// TIA Portal project "THAY PHUONG" (V17)

(* hardware
DEVICE "S7-1200 station_1"  S7-1200 Station
   slot 0: "Rack_0"  S7-1200 Rack  Rack  V1.0
   slot 1: "PLC_1"  CPU 1214C DC/DC/DC  6ES7 214-1AG40-0XB0  V4.0
*)

// ===== PLC "PLC_1"  CPU 1214C DC/DC/DC =====

VAR_GLOBAL   // PLC tag table "Default tag table"
   "System_Byte" AT %MB100 : Byte;
   "FirstScan" AT %M100.0 : Bool;
   "DiagStatusUpdate" AT %M100.1 : Bool;
   "AlwaysTRUE" AT %M100.2 : Bool;
   "AlwaysFALSE" AT %M100.3 : Bool;
   "Clock_Byte" AT %MB200 : Byte;
   "Clock_10Hz" AT %M200.0 : Bool;
   "Clock_5Hz" AT %M200.1 : Bool;
   "Clock_2.5Hz" AT %M200.2 : Bool;
   "Clock_2Hz" AT %M200.3 : Bool;
   "Clock_1.25Hz" AT %M200.4 : Bool;
   "Clock_1Hz" AT %M200.5 : Bool;
   "Clock_0.625Hz" AT %M200.6 : Bool;
   "Clock_0.5Hz" AT %M200.7 : Bool;
   "System_Byte(1)" AT %MB100 : Byte;
   "System_Byte(2)" AT %MB0 : Byte;
   "System_Byte(3)" AT %MB0 : Byte;
END_VAR

VAR_GLOBAL   // PLC tag table "STEP"
   "STEP1" AT %M0.0 : Bool;
   "STEP2" AT %M0.1 : Bool;
   "STEP3" AT %M0.2 : Bool;
   "STEP4" AT %M0.3 : Bool;
   "STEP5" AT %M0.4 : Bool;
   "STEP6" AT %M0.5 : Bool;
   "STEP7" AT %M0.6 : Bool;
   "STEP8" AT %M0.7 : Bool;
   "STEP9" AT %M1.0 : Bool;
   "STEP10" AT %M1.1 : Bool;
   "STEP11" AT %M1.2 : Bool;
END_VAR

VAR_GLOBAL   // PLC tag table "OUTPUT"
   "H1" AT %Q0.0 : Bool;
   "H2" AT %Q0.1 : Bool;
   "H3" AT %Q0.2 : Bool;
   "H4" AT %Q0.3 : Bool;
   "H5" AT %Q0.4 : Bool;
   "H6" AT %Q0.5 : Bool;
   "H7" AT %Q0.6 : Bool;
   "H8" AT %Q0.7 : Bool;
END_VAR

VAR_GLOBAL   // PLC tag table "iNPUT"
   "B1" AT %I0.0 : Bool;
   "B2" AT %I0.1 : Bool;
   "B3" AT %I0.2 : Bool;
   "S1" AT %I0.3 : Bool;
   "S2" AT %I0.4 : Bool;
   "S6n" AT %I0.5 : Bool;
   "S7n" AT %I0.6 : Bool;
   "S8" AT %I0.7 : Bool;
END_VAR

// folder: System blocks/Program resources

DATA_BLOCK "T1"   // DB1
{ S7_Optimized_Access := 'TRUE' }
AUTHOR : Simatic
FAMILY : IEC
NAME : IEC_TMR
VERSION : 1.0
// stored: InstanceOfName IEC_TIMER
"IEC_TIMER"
BEGIN
END_DATA_BLOCK

DATA_BLOCK "T2"   // DB2
{ S7_Optimized_Access := 'TRUE' }
AUTHOR : Simatic
FAMILY : IEC
NAME : IEC_TMR
VERSION : 1.0
// stored: InstanceOfName IEC_TIMER
"IEC_TIMER"
BEGIN
END_DATA_BLOCK

DATA_BLOCK "TimerH1"   // DB3
{ S7_Optimized_Access := 'TRUE' }
AUTHOR : Simatic
FAMILY : IEC
NAME : IEC_TMR
VERSION : 1.0
// stored: InstanceOfName IEC_TIMER
"IEC_TIMER"
BEGIN
END_DATA_BLOCK

DATA_BLOCK "TimerH2"   // DB4
{ S7_Optimized_Access := 'TRUE' }
AUTHOR : Simatic
FAMILY : IEC
NAME : IEC_TMR
VERSION : 1.0
// stored: InstanceOfName IEC_TIMER
"IEC_TIMER"
BEGIN
END_DATA_BLOCK

DATA_BLOCK "TimerH2B"   // DB5
{ S7_Optimized_Access := 'TRUE' }
AUTHOR : Simatic
FAMILY : IEC
NAME : IEC_TMR
VERSION : 1.0
// stored: InstanceOfName IEC_TIMER
"IEC_TIMER"
BEGIN
END_DATA_BLOCK

DATA_BLOCK "Timer1"   // DB6
{ S7_Optimized_Access := 'TRUE' }
AUTHOR : Simatic
FAMILY : IEC
NAME : IEC_TMR
VERSION : 1.0
// stored: InstanceOfName IEC_TIMER
"IEC_TIMER"
BEGIN
END_DATA_BLOCK

DATA_BLOCK "Timer2"   // DB7
{ S7_Optimized_Access := 'TRUE' }
AUTHOR : Simatic
FAMILY : IEC
NAME : IEC_TMR
VERSION : 1.0
// stored: InstanceOfName IEC_TIMER
"IEC_TIMER"
BEGIN
END_DATA_BLOCK

// folder: (top level)

FUNCTION "BAI1" : Void   // FC1, FBD
{ S7_Optimized_Access := 'TRUE' }
VERSION : 0.1
BEGIN

REGION Network 1
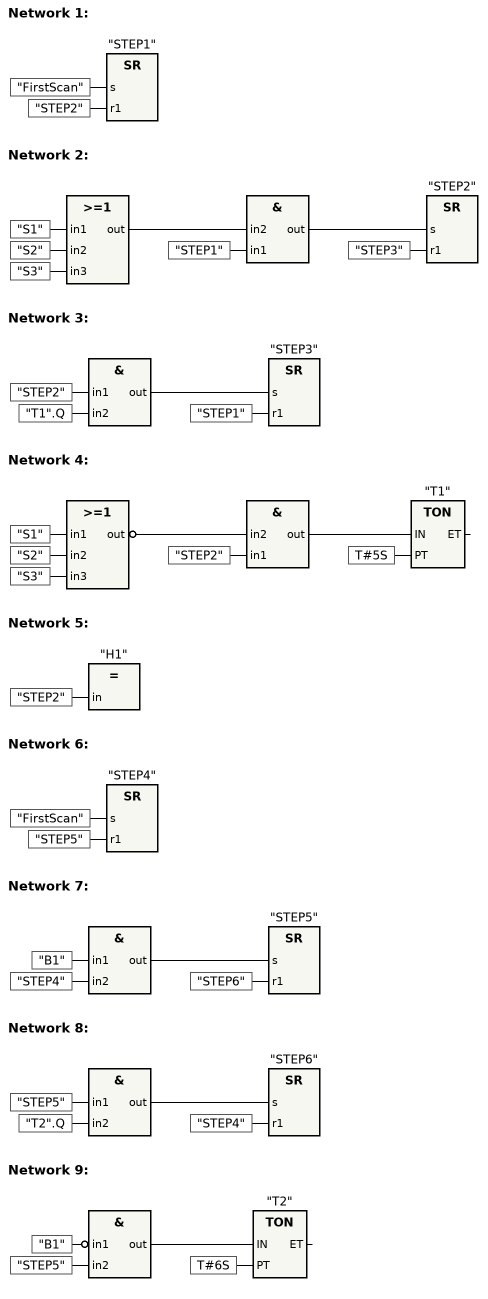
   IF "FirstScan" THEN
       "STEP1" := TRUE;   // SR flip-flop
   END_IF;
   IF "STEP2" THEN "STEP1" := FALSE; END_IF;
END_REGION

REGION Network 2
   IF ("S1" OR "S2" OR "S3") AND "STEP1" THEN
       "STEP2" := TRUE;   // SR flip-flop
   END_IF;
   IF "STEP3" THEN "STEP2" := FALSE; END_IF;
END_REGION

REGION Network 3
   IF "STEP2" AND "T1".Q THEN
       "STEP3" := TRUE;   // SR flip-flop
   END_IF;
   IF "STEP1" THEN "STEP3" := FALSE; END_IF;
END_REGION

REGION Network 4
   "T1".TON(IN := NOT ("S1" OR "S2" OR "S3") AND "STEP2", PT := T#5S);
END_REGION

REGION Network 5
   "H1" := "STEP2";
END_REGION

REGION Network 6
   IF "FirstScan" THEN
       "STEP4" := TRUE;   // SR flip-flop
   END_IF;
   IF "STEP5" THEN "STEP4" := FALSE; END_IF;
END_REGION

REGION Network 7
   IF "B1" AND "STEP4" THEN
       "STEP5" := TRUE;   // SR flip-flop
   END_IF;
   IF "STEP6" THEN "STEP5" := FALSE; END_IF;
END_REGION

REGION Network 8
   IF "STEP5" AND "T2".Q THEN
       "STEP6" := TRUE;   // SR flip-flop
   END_IF;
   IF "STEP4" THEN "STEP6" := FALSE; END_IF;
END_REGION

REGION Network 9
   "T2".TON(IN := NOT "B1" AND "STEP5", PT := T#6S);
END_REGION

REGION Network 10
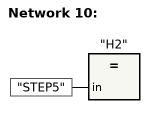
   "H2" := "STEP5";
END_REGION
END_FUNCTION

FUNCTION "HunqD_De1" : Void   // FC2, FBD
{ S7_Optimized_Access := 'TRUE' }
VERSION : 0.1
BEGIN

REGION Network 1: STEP 1
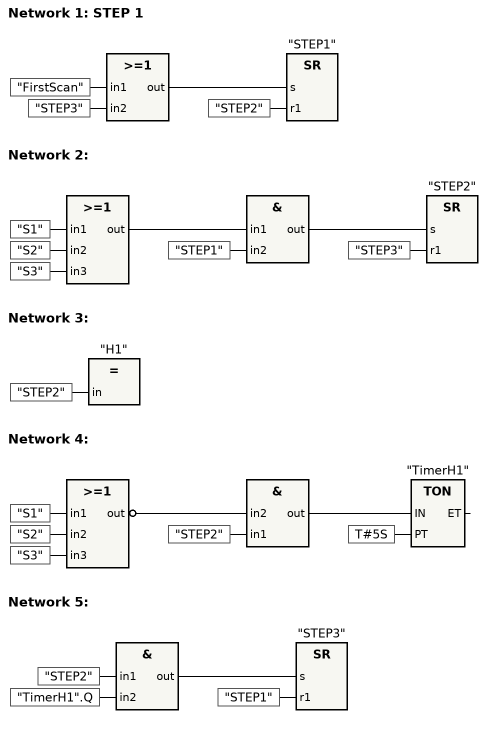
   IF "FirstScan" OR "STEP3" THEN
       "STEP1" := TRUE;   // SR flip-flop
   END_IF;
   IF "STEP2" THEN "STEP1" := FALSE; END_IF;
END_REGION

REGION Network 2
   IF ("S1" OR "S2" OR "S3") AND "STEP1" THEN
       "STEP2" := TRUE;   // SR flip-flop
   END_IF;
   IF "STEP3" THEN "STEP2" := FALSE; END_IF;
END_REGION

REGION Network 3
   "H1" := "STEP2";
END_REGION

REGION Network 4
   "TimerH1".TON(IN := NOT ("S1" OR "S2" OR "S3") AND "STEP2", PT := T#5S);
END_REGION

REGION Network 5
   IF "STEP2" AND "TimerH1".Q THEN
       "STEP3" := TRUE;   // SR flip-flop
   END_IF;
   IF "STEP1" THEN "STEP3" := FALSE; END_IF;
END_REGION
END_FUNCTION

FUNCTION "HunqD_De2" : Void   // FC2, FBD
{ S7_Optimized_Access := 'TRUE' }
VERSION : 0.1
BEGIN

REGION Network 1: STEP 1
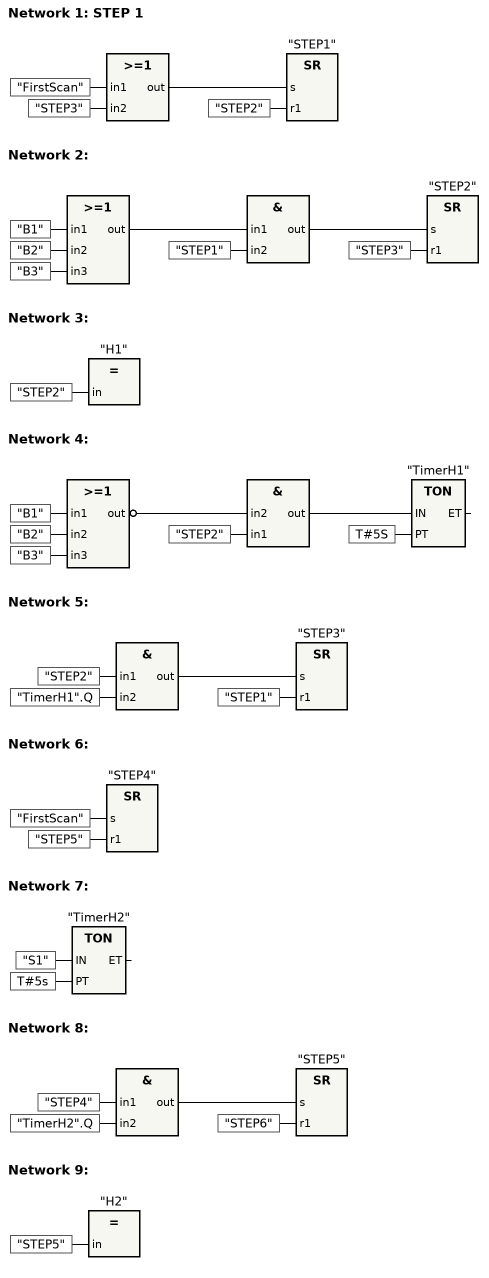
   IF "FirstScan" OR "STEP3" THEN
       "STEP1" := TRUE;   // SR flip-flop
   END_IF;
   IF "STEP2" THEN "STEP1" := FALSE; END_IF;
END_REGION

REGION Network 2
   IF ("B1" OR "B2" OR "B3") AND "STEP1" THEN
       "STEP2" := TRUE;   // SR flip-flop
   END_IF;
   IF "STEP3" THEN "STEP2" := FALSE; END_IF;
END_REGION

REGION Network 3
   "H1" := "STEP2";
END_REGION

REGION Network 4
   "TimerH1".TON(IN := NOT ("B1" OR "B2" OR "B3") AND "STEP2", PT := T#5S);
END_REGION

REGION Network 5
   IF "STEP2" AND "TimerH1".Q THEN
       "STEP3" := TRUE;   // SR flip-flop
   END_IF;
   IF "STEP1" THEN "STEP3" := FALSE; END_IF;
END_REGION

REGION Network 6
   IF "FirstScan" THEN
       "STEP4" := TRUE;   // SR flip-flop
   END_IF;
   IF "STEP5" THEN "STEP4" := FALSE; END_IF;
END_REGION

REGION Network 7
   "TimerH2".TON(IN := "S1", PT := T#5s);
END_REGION

REGION Network 8
   IF "STEP4" AND "TimerH2".Q THEN
       "STEP5" := TRUE;   // SR flip-flop
   END_IF;
   IF "STEP6" THEN "STEP5" := FALSE; END_IF;
END_REGION

REGION Network 9
   "H2" := "STEP5";
END_REGION

REGION Network 10
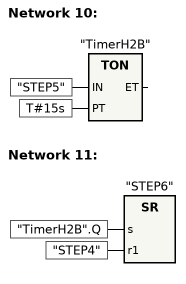
   "TimerH2B".TON(IN := "STEP5", PT := T#15s);
END_REGION

REGION Network 11
   IF "TimerH2B".Q THEN
       "STEP6" := TRUE;   // SR flip-flop
   END_IF;
   IF "STEP4" THEN "STEP6" := FALSE; END_IF;
END_REGION
END_FUNCTION

FUNCTION "HunqD_De3" : Void   // FC3, FBD
{ S7_Optimized_Access := 'TRUE' }
VERSION : 0.1
BEGIN

REGION Network 1
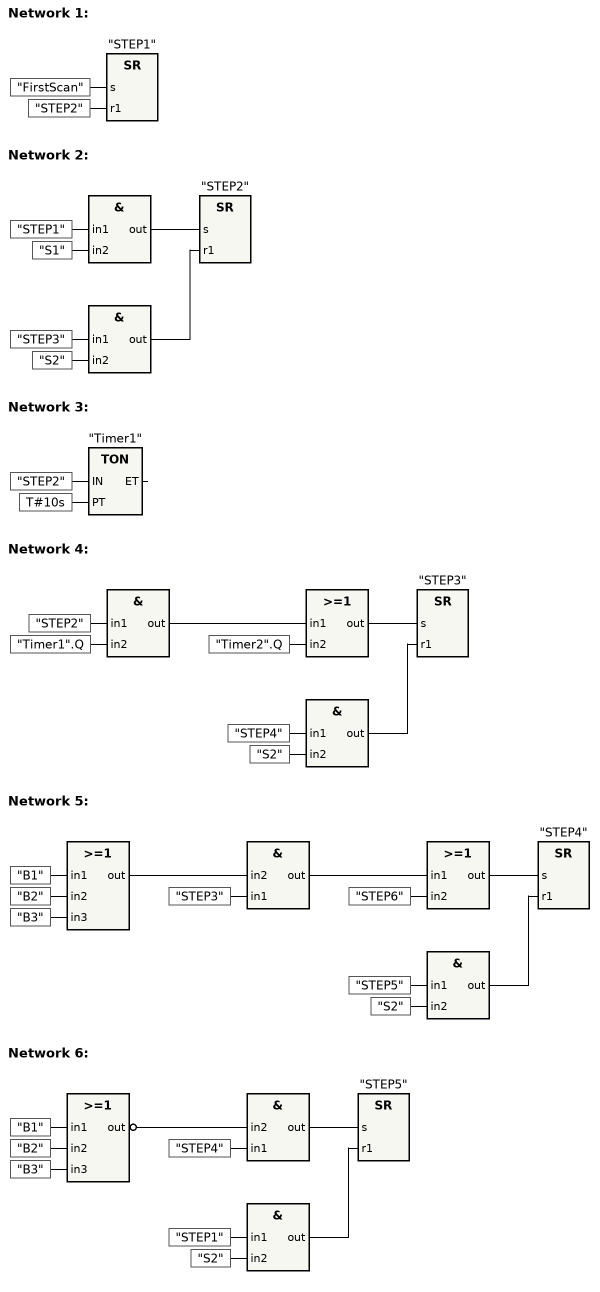
   IF "FirstScan" THEN
       "STEP1" := TRUE;   // SR flip-flop
   END_IF;
   IF "STEP2" THEN "STEP1" := FALSE; END_IF;
END_REGION

REGION Network 2
   IF "STEP1" AND "S1" THEN
       "STEP2" := TRUE;   // SR flip-flop
   END_IF;
   IF "STEP3" AND "S2" THEN "STEP2" := FALSE; END_IF;
END_REGION

REGION Network 3
   "Timer1".TON(IN := "STEP2", PT := T#10s);
END_REGION

REGION Network 4
   IF ("STEP2" AND "Timer1".Q) OR "Timer2".Q THEN
       "STEP3" := TRUE;   // SR flip-flop
   END_IF;
   IF "STEP4" AND "S2" THEN "STEP3" := FALSE; END_IF;
END_REGION

REGION Network 5
   IF (("B1" OR "B2" OR "B3") AND "STEP3") OR "STEP6" THEN
       "STEP4" := TRUE;   // SR flip-flop
   END_IF;
   IF "STEP5" AND "S2" THEN "STEP4" := FALSE; END_IF;
END_REGION

REGION Network 6
   IF NOT ("B1" OR "B2" OR "B3") AND "STEP4" THEN
       "STEP5" := TRUE;   // SR flip-flop
   END_IF;
   IF "STEP1" AND "S2" THEN "STEP5" := FALSE; END_IF;
END_REGION

REGION Network 7
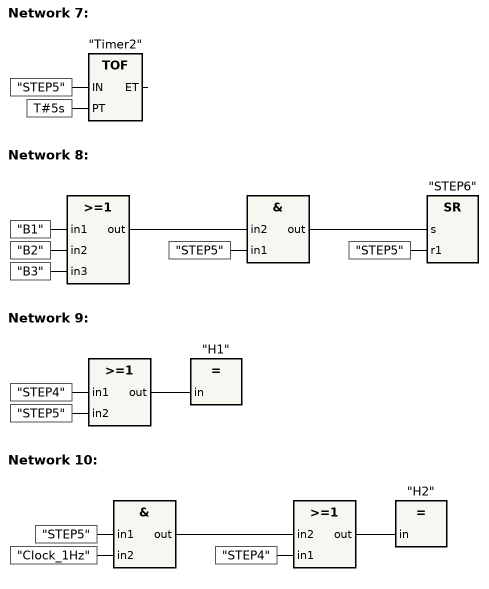
   "Timer2".TOF(IN := "STEP5", PT := T#5s);
END_REGION

REGION Network 8
   IF ("B1" OR "B2" OR "B3") AND "STEP5" THEN
       "STEP6" := TRUE;   // SR flip-flop
   END_IF;
   IF "STEP5" THEN "STEP6" := FALSE; END_IF;
END_REGION

REGION Network 9
   "H1" := "STEP4" OR "STEP5";
END_REGION

REGION Network 10
   "H2" := ("STEP5" AND "Clock_1Hz") OR "STEP4";
END_REGION
END_FUNCTION

ORGANIZATION_BLOCK "Main"   // OB1, LAD, ProgramCycle
TITLE = "Main Program Sweep (Cycle)"
{ S7_Optimized_Access := 'TRUE' }
VERSION : 0.1
   VAR_INPUT
      Initial_Call : Bool;   // Initial call of this OB
      Remanence : Bool;   // =True, if remanent data are available
   END_VAR
BEGIN

REGION Network 1
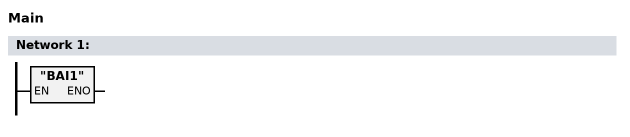
   RUNG wire#powerrail
      "BAI1"()
   END_RUNG
   // the same network as SCL:
   "BAI1"();
END_REGION
END_ORGANIZATION_BLOCK